// TwinCAT 3 PLC project Example
// ProgramVersion: 3.1.4023.0
// libraries:
//   Tc2_Math, * (Beckhoff Automation GmbH)
//   Tc2_Standard, * (Beckhoff Automation GmbH)
//   Tc2_System, * (Beckhoff Automation GmbH)
//   Tc3_Module, * (Beckhoff Automation GmbH)
// project tree:
//   DUTs/Enums/ E_Error.TcDUT
//   GVLs/ Param_Constants.TcGVL
//   ITFs/Core/ I_Object.TcIO, I_Operator.TcIO
//   ITFs/ I_Scalar.TcIO, I_Vector.TcIO
//   ITFs/Operators/ I_Addition.TcIO, I_Division.TcIO, I_Multiplication.TcIO, I_Subtraction.TcIO
//   / PlcTask.TcTTO
//   POUs/FunctionBlock/ FB_Scalar.TcPOU, FB_Vector.TcPOU
//   POUs/ MAIN.TcPOU
// real-time tasks:
//   TASK PlcTask: cycle T#10ms, priority 20, ADS port 350

CONFIGURATION Example
    RESOURCE PLC ON TwinCAT3
        TASK PlcTask(INTERVAL := T#10ms, PRIORITY := 20);
        PROGRAM MAIN WITH PlcTask : MAIN;
    END_RESOURCE
END_CONFIGURATION

// ---- DUTs/Enums/E_Error.TcDUT
{attribute 'qualified_only'}
{attribute 'strict'}
{attribute 'to_string'}
TYPE E_Error :
(
	NoError := 0,
	IntegerOverflow := 10,
	NaN,
	PositiveInfinity,
	NegativeInfinity,
	Truncation,
	TypeMismatch := 100
)BYTE;
END_TYPE

// ---- GVLs/Param_Constants.TcGVL
{attribute 'qualified_only'}
VAR_GLOBAL CONSTANT
	QR_CODE_LENGTH : __UXINT := 4;
END_VAR

// ---- ITFs/Core/I_Object.TcIO
// Base interface for an object.
INTERFACE I_Object EXTENDS __SYSTEM.IQueryInterface

END_INTERFACE

// ---- ITFs/Core/I_Operator.TcIO
// Base interface for an operator.
INTERFACE I_Operator EXTENDS I_Object

END_INTERFACE

// ---- ITFs/I_Scalar.TcIO
INTERFACE I_Scalar EXTENDS I_Object

METHOD ToF64 : LREAL
VAR_OUTPUT
	e : E_Error;
END_VAR
END_METHOD

METHOD ToI64 : LINT
VAR_OUTPUT
	e : E_Error;
END_VAR
END_METHOD

METHOD ToU8 : BYTE
VAR_OUTPUT
	e : E_Error;
END_VAR
END_METHOD

END_INTERFACE

// ---- ITFs/I_Vector.TcIO
INTERFACE I_Vector EXTENDS I_Object

METHOD ToArray : ARRAY[0..2] OF LREAL
VAR_INPUT
END_VAR
END_METHOD

PROPERTY X : LREAL
GET
END_GET
SET
END_SET
END_PROPERTY

PROPERTY Y : LREAL
GET
END_GET
SET
END_SET
END_PROPERTY

PROPERTY Z : LREAL
GET
END_GET
SET
END_SET
END_PROPERTY

END_INTERFACE

// ---- ITFs/Operators/I_Addition.TcIO
INTERFACE I_Addition EXTENDS I_Operator

METHOD Plus : I_Addition
VAR_INPUT
	ipObject : I_Object;
END_VAR
VAR_OUTPUT
	e : E_Error;
END_VAR
END_METHOD

END_INTERFACE

// ---- ITFs/Operators/I_Division.TcIO
INTERFACE I_Division EXTENDS I_Operator

METHOD DivideBy : I_Division
VAR_INPUT
	ipObject : I_Object;
END_VAR
VAR_OUTPUT
	e : E_Error;
END_VAR
END_METHOD

END_INTERFACE

// ---- ITFs/Operators/I_Multiplication.TcIO
INTERFACE I_Multiplication EXTENDS I_Operator

METHOD Times : I_Multiplication
VAR_INPUT
	ipObject : I_Object;
END_VAR
VAR_OUTPUT
	e : E_Error;
END_VAR
END_METHOD

END_INTERFACE

// ---- ITFs/Operators/I_Subtraction.TcIO
INTERFACE I_Subtraction EXTENDS I_Operator

METHOD Minus : I_Subtraction
VAR_INPUT
	ipObject : I_Object;
END_VAR
VAR_OUTPUT
	e : E_Error;
END_VAR
END_METHOD

END_INTERFACE

// ---- POUs/MAIN.TcPOU
PROGRAM MAIN
VAR
	bDoubleSquareScal, bAddVec, bCrossProd, bScaleVec: BOOL;
	eError : E_Error;
	fbScalar : FB_Scalar(2.2);
	fbVec1 : FB_Vector(1,2,3);
	fbVec2 : FB_Vector(3,2,1);
END_VAR

IF bDoubleSquareScal THEN 
	bDoubleSquareScal := FALSE;
	fbScalar.Times(fbScalar.Plus(fbScalar));
	END_IF

IF bAddVec THEN
	bAddVec := FALSE;
	fbVec1.Plus(fbVec2);
	END_IF
	
IF bCrossProd THEN
	bCrossProd := FALSE;
	fbVec1.Times(fbVec2);
	END_IF
	
IF bScaleVec THEN
	bScaleVec := FALSE;
	fbVec1.Times(fbScalar);
	END_IF

END_PROGRAM

// ---- POUs/FunctionBlock/FB_Scalar.TcPOU
{attribute 'no_explicit_call' := 'do not call this function block directly'}
FUNCTION_BLOCK FB_Scalar IMPLEMENTS I_Scalar, I_Addition, I_Subtraction, I_Multiplication, I_Division
VAR
	_fValue : LREAL; 
END_VAR

METHOD DivideBy : I_Division
VAR_INPUT
	ipObject : I_Object;
END_VAR
VAR_OUTPUT
	e : E_Error;
END_VAR
VAR
	Tmp : LREAL;
	ipNumber : I_Scalar;
END_VAR
DivideBy := THIS^;

IF NOT __QUERYINTERFACE(ipObject, ipNumber) THEN e := E_Error.TypeMismatch; RETURN; END_IF

Tmp := ipNumber.ToF64(e => e);
IF Tmp = 0 THEN 
	THIS^._fValue := SEL(Tmp > 0, -1*TO_LREAL('#Inf'), TO_LREAL('#Inf'));
	RETURN;
	END_IF

IF e <> E_Error.NoError THEN 
	THIS^._fValue := ipNumber.ToF64();
	END_IF

THIS^._fValue := THIS^.ToF64() / ipNumber.ToF64();
END_METHOD

{attribute 'hide'}
METHOD FB_init : BOOL
VAR_INPUT
	bInitRetains : BOOL; // if TRUE, the retain variables are initialized (warm start / cold start)
	bInCopyCode : BOOL;  // if TRUE, the instance afterwards gets moved into the copy code (online change)
	fInitValue : LREAL;
END_VAR
THIS^._fValue := fInitValue;
END_METHOD

METHOD Minus : I_Subtraction
VAR_INPUT
	ipObject : I_Object;
END_VAR
VAR_OUTPUT
	e : E_Error;
END_VAR
VAR
	e1, e2 : E_Error;
	ipNumber : I_Scalar;
END_VAR
Minus := THIS^;

IF NOT __QUERYINTERFACE(ipObject, ipNumber) THEN e := E_Error.TypeMismatch; RETURN; END_IF

THIS^._fValue := THIS^.ToF64(e => e1) - ipNumber.ToF64(e => e2);

e := MAX(e1, e2);
END_METHOD

METHOD Plus : I_Addition
VAR_INPUT
	ipObject : I_Object;
END_VAR
VAR_OUTPUT
	e : E_Error;
END_VAR
VAR
	e1, e2 : E_Error;
	ipNumber : I_Scalar;
END_VAR
Plus := THIS^;

IF NOT __QUERYINTERFACE(ipObject, ipNumber) THEN e := E_Error.TypeMismatch; RETURN; END_IF

THIS^._fValue := THIS^.ToF64(e => e1) + ipNumber.ToF64(e => e2);

e := MAX(e1, e2);
END_METHOD

METHOD SetValue : REFERENCE TO FB_Scalar
VAR_INPUT
	fValue : LREAL;
END_VAR
SetValue REF= THIS^;

THIS^._fValue := fValue;
END_METHOD

METHOD Times : I_Multiplication
VAR_INPUT
	ipObject : I_Object;
END_VAR
VAR_OUTPUT
	e : E_Error;
END_VAR
VAR
	e1, e2 : E_Error;
	ipNumber : I_Scalar;
END_VAR
Times := THIS^;

IF NOT __QUERYINTERFACE(ipObject, ipNumber) THEN e := E_Error.TypeMismatch; RETURN; END_IF

THIS^._fValue := THIS^.ToF64(e => e1) * ipNumber.ToF64( e => e2);

e := MAX(e1, e2);
END_METHOD

METHOD ToF64 : LREAL
VAR_OUTPUT
	e	: E_Error;
END_VAR
ToF64 := THIS^._fValue;

IF TO_STRING(THIS^._fValue) = '#NaN' THEN 
	e := E_Error.NaN;
ELSIF TO_STRING(THIS^._fValue) = '#Inf' THEN
	e := E_Error.PositiveInfinity;
ELSIF TO_STRING(THIS^._fValue) = '-#Inf' THEN
	e := E_Error.NegativeInfinity;
	END_IF
END_METHOD

METHOD ToI64 : LINT
VAR_OUTPUT
	e	: E_Error;
END_VAR
ToI64 := TO_LINT(THIS^._fValue);

// Check for truncation.
IF Tc2_Math.FRAC(THIS^._fValue) <> 0  THEN 
	e := E_Error.Truncation;
	END_IF
END_METHOD

METHOD ToU8 : BYTE
VAR_OUTPUT
	e	: E_Error;
END_VAR
ToU8 := TO_BYTE(THIS^._fValue);

// Check for truncation.
IF Tc2_Math.FRAC(THIS^._fValue) <> 0  THEN 
	e := E_Error.Truncation;
	END_IF

// Bounds check.
IF THIS^._fValue < 0 OR THIS^._fValue > 255 THEN 
	e := E_Error.IntegerOverflow;
	END_IF
END_METHOD

END_FUNCTION_BLOCK

// ---- POUs/FunctionBlock/FB_Vector.TcPOU
{attribute 'no_explicit_call' := 'do not call this function block directly'}
FUNCTION_BLOCK FB_Vector IMPLEMENTS I_Vector, I_Addition, I_Subtraction, I_Multiplication
VAR
	_fX, _fY, _fZ : LREAL;
END_VAR

{attribute 'hide'}
METHOD FB_init : BOOL
VAR_INPUT
	bInitRetains : BOOL; // if TRUE, the retain variables are initialized (warm start / cold start)
	bInCopyCode : BOOL;  // if TRUE, the instance afterwards gets moved into the copy code (online change)
	fX, fY, fZ : LREAL;
END_VAR
THIS^.SetValue(fX, fY, fZ);
END_METHOD

METHOD Minus : I_Subtraction
VAR_INPUT
	ipObject : I_Object;
END_VAR
VAR_OUTPUT
	e : E_Error;
END_VAR
VAR
	ipVector : I_Vector;
END_VAR
Minus := THIS^;

IF NOT __QUERYINTERFACE(ipObject, ipVector) THEN e := E_Error.TypeMismatch; RETURN; END_IF

THIS^._fX := THIS^._fX - ipVector.X;
THIS^._fY := THIS^._fY - ipVector.Y;
THIS^._fZ := THIS^._fZ - ipVector.Z;
END_METHOD

METHOD Plus : I_Addition
VAR_INPUT
	ipObject : I_Object;
END_VAR
VAR_OUTPUT
	e : E_Error;
END_VAR
VAR
	ipVector : I_Vector;
END_VAR
Plus := THIS^;

IF NOT __QUERYINTERFACE(ipObject, ipVector) THEN e := E_Error.TypeMismatch; RETURN; END_IF

THIS^._fX := THIS^._fX + ipVector.X;
THIS^._fY := THIS^._fY + ipVector.Y;
THIS^._fZ := THIS^._fZ + ipVector.Z;
END_METHOD

METHOD SetValue : REFERENCE TO FB_Vector
VAR_INPUT
	fX, fY, fZ : LREAL;
END_VAR
SetValue REF= THIS^;

THIS^._fX := fX;
THIS^._fY := fY;
THIS^._fZ := fZ;
END_METHOD

METHOD Times : I_Multiplication
VAR_INPUT
	ipObject : I_Object;
END_VAR
VAR_OUTPUT
	e : E_Error;
END_VAR
VAR
	ipNumber : I_Scalar;
	ipVector : I_Vector;
	TmpX, TmpY, TmpZ : LREAL;
END_VAR
Times := THIS^;

// Scale vector.
IF __QUERYINTERFACE(ipObject, ipNumber) THEN 
	THIS^.SetValue( THIS^._fX * ipNumber.ToF64(),
					THIS^._fY * ipNumber.ToF64(),
					THIS^._fZ * ipNumber.ToF64());
	RETURN;
	END_IF

// Do the cross-product.
IF __QUERYINTERFACE(ipObject, ipVector) THEN 
	TmpX := THIS^._fX; TmpY := THIS^._fY; TmpZ := THIS^._fZ;
	THIS^.SetValue(	(TmpY*ipVector.Z) - (TmpZ*ipVector.Y),
					(TmpZ*ipVector.X) - (TmpX*ipVector.Y),
					(TmpX*ipVector.Y) - (TmpY*ipVector.X));
	
	RETURN; 
	END_IF

e := E_Error.TypeMismatch;
END_METHOD

METHOD ToArray : ARRAY[0..2] OF LREAL
VAR_INPUT
END_VAR
ToArray[0]:= THIS^._fX;
ToArray[1]:= THIS^._fY;
ToArray[2]:= THIS^._fZ;
END_METHOD

PROPERTY X : LREAL
GET
X := THIS^._fX;
END_GET
SET
THIS^._fX := X;
END_SET
END_PROPERTY

PROPERTY Y : LREAL
GET
Y := THIS^._fY;
END_GET
SET
THIS^._fY:= Y;
END_SET
END_PROPERTY

PROPERTY Z : LREAL
GET
Z := THIS^._fZ;
END_GET
SET
THIS^._fZ := Z;
END_SET
END_PROPERTY

END_FUNCTION_BLOCK
